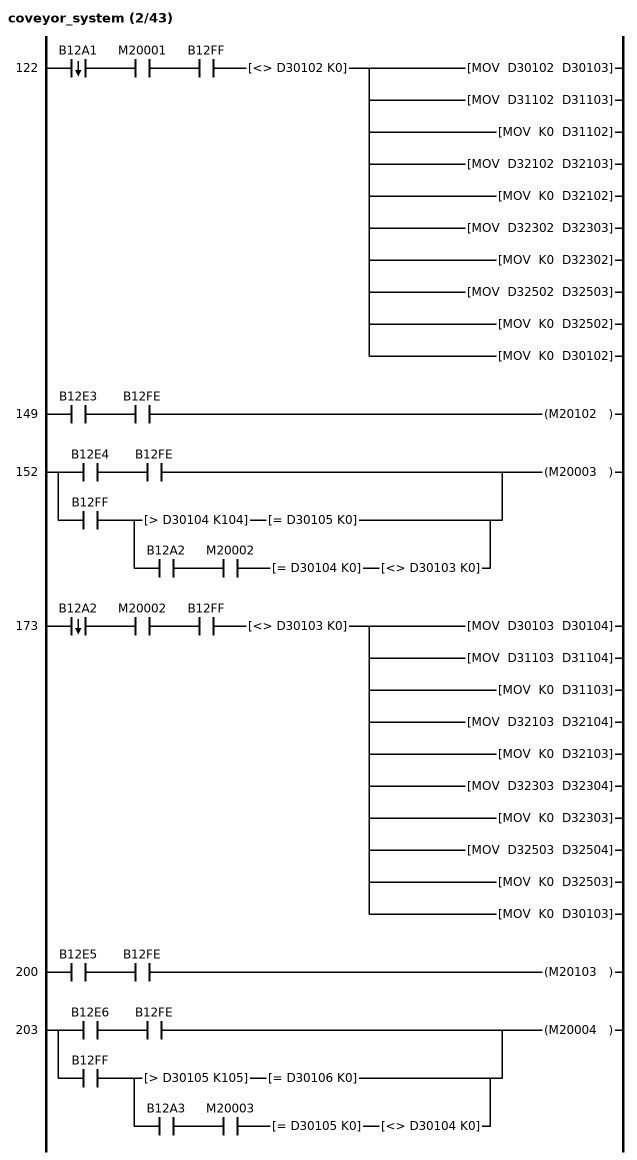
[picture p168: ladder of coveyor_system, rungs at steps 122 to 203]
122   LDF     B12A1
      AND     M20001
      AND     B12FF
      AND<>   D30102 K0
      MOV     D30102 D30103
      MOV     D31102 D31103
      MOV     K0 D31102
      MOV     D32102 D32103
      MOV     K0 D32102
      MOV     D32302 D32303
      MOV     K0 D32302
      MOV     D32502 D32503
      MOV     K0 D32502
      MOV     K0 D30102
149   LD      B12E3
      AND     B12FE
      OUT     M20102
152   LD      B12E4
      AND     B12FE
      LD      B12FF
      LD>     D30104 K104
      AND=    D30105 K0
      LD      B12A2
      AND     M20002
      AND=    D30104 K0
      AND<>   D30103 K0
      ORB
      ANB
      ORB
      OUT     M20003
173   LDF     B12A2
      AND     M20002
      AND     B12FF
      AND<>   D30103 K0
      MOV     D30103 D30104
      MOV     D31103 D31104
      MOV     K0 D31103
      MOV     D32103 D32104
      MOV     K0 D32103
      MOV     D32303 D32304
      MOV     K0 D32303
      MOV     D32503 D32504
      MOV     K0 D32503
      MOV     K0 D30103
200   LD      B12E5
      AND     B12FE
      OUT     M20103
203   LD      B12E6
      AND     B12FE
      LD      B12FF
      LD>     D30105 K105
      AND=    D30106 K0
      LD      B12A3
      AND     M20003
      AND=    D30105 K0
      AND<>   D30104 K0
      ORB
      ANB
      ORB
      OUT     M20004
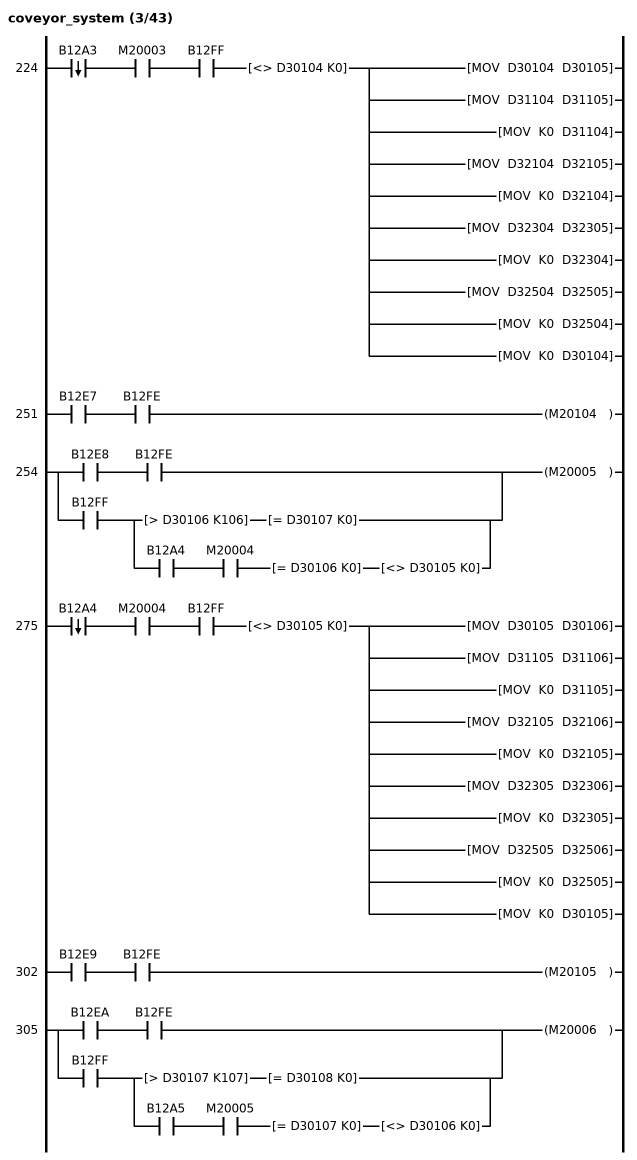
224   LDF     B12A3
      AND     M20003
      AND     B12FF
      AND<>   D30104 K0
      MOV     D30104 D30105
      MOV     D31104 D31105
      MOV     K0 D31104
      MOV     D32104 D32105
      MOV     K0 D32104
      MOV     D32304 D32305
      MOV     K0 D32304
      MOV     D32504 D32505
      MOV     K0 D32504
      MOV     K0 D30104
251   LD      B12E7
      AND     B12FE
      OUT     M20104
254   LD      B12E8
      AND     B12FE
      LD      B12FF
      LD>     D30106 K106
      AND=    D30107 K0
      LD      B12A4
      AND     M20004
      AND=    D30106 K0
      AND<>   D30105 K0
      ORB
      ANB
      ORB
      OUT     M20005
275   LDF     B12A4
      AND     M20004
      AND     B12FF
      AND<>   D30105 K0
      MOV     D30105 D30106
      MOV     D31105 D31106
      MOV     K0 D31105
      MOV     D32105 D32106
      MOV     K0 D32105
      MOV     D32305 D32306
      MOV     K0 D32305
      MOV     D32505 D32506
      MOV     K0 D32505
      MOV     K0 D30105
302   LD      B12E9
      AND     B12FE
      OUT     M20105
305   LD      B12EA
      AND     B12FE
      LD      B12FF
      LD>     D30107 K107
      AND=    D30108 K0
      LD      B12A5
      AND     M20005
      AND=    D30107 K0
      AND<>   D30106 K0
      ORB
      ANB
      ORB
      OUT     M20006
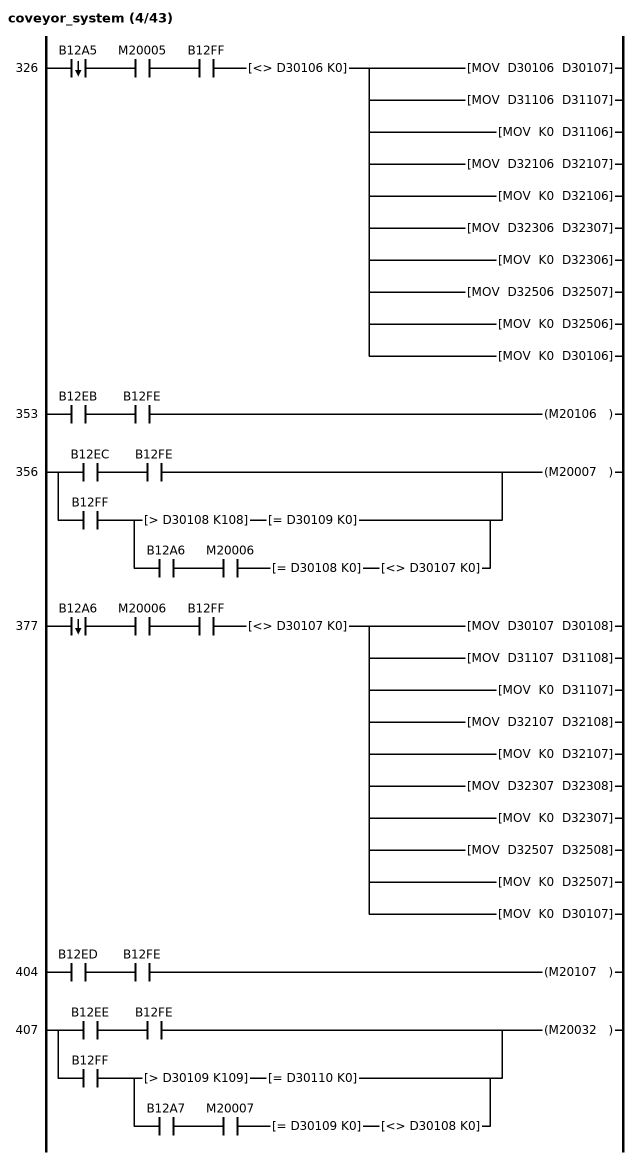
326   LDF     B12A5
      AND     M20005
      AND     B12FF
      AND<>   D30106 K0
      MOV     D30106 D30107
      MOV     D31106 D31107
      MOV     K0 D31106
      MOV     D32106 D32107
      MOV     K0 D32106
      MOV     D32306 D32307
      MOV     K0 D32306
      MOV     D32506 D32507
      MOV     K0 D32506
      MOV     K0 D30106
353   LD      B12EB
      AND     B12FE
      OUT     M20106
356   LD      B12EC
      AND     B12FE
      LD      B12FF
      LD>     D30108 K108
      AND=    D30109 K0
      LD      B12A6
      AND     M20006
      AND=    D30108 K0
      AND<>   D30107 K0
      ORB
      ANB
      ORB
      OUT     M20007
377   LDF     B12A6
      AND     M20006
      AND     B12FF
      AND<>   D30107 K0
      MOV     D30107 D30108
      MOV     D31107 D31108
      MOV     K0 D31107
      MOV     D32107 D32108
      MOV     K0 D32107
      MOV     D32307 D32308
      MOV     K0 D32307
      MOV     D32507 D32508
      MOV     K0 D32507
      MOV     K0 D30107
404   LD      B12ED
      AND     B12FE
      OUT     M20107
407   LD      B12EE
      AND     B12FE
      LD      B12FF
      LD>     D30109 K109
      AND=    D30110 K0
      LD      B12A7
      AND     M20007
      AND=    D30109 K0
      AND<>   D30108 K0
      ORB
      ANB
      ORB
      OUT     M20032
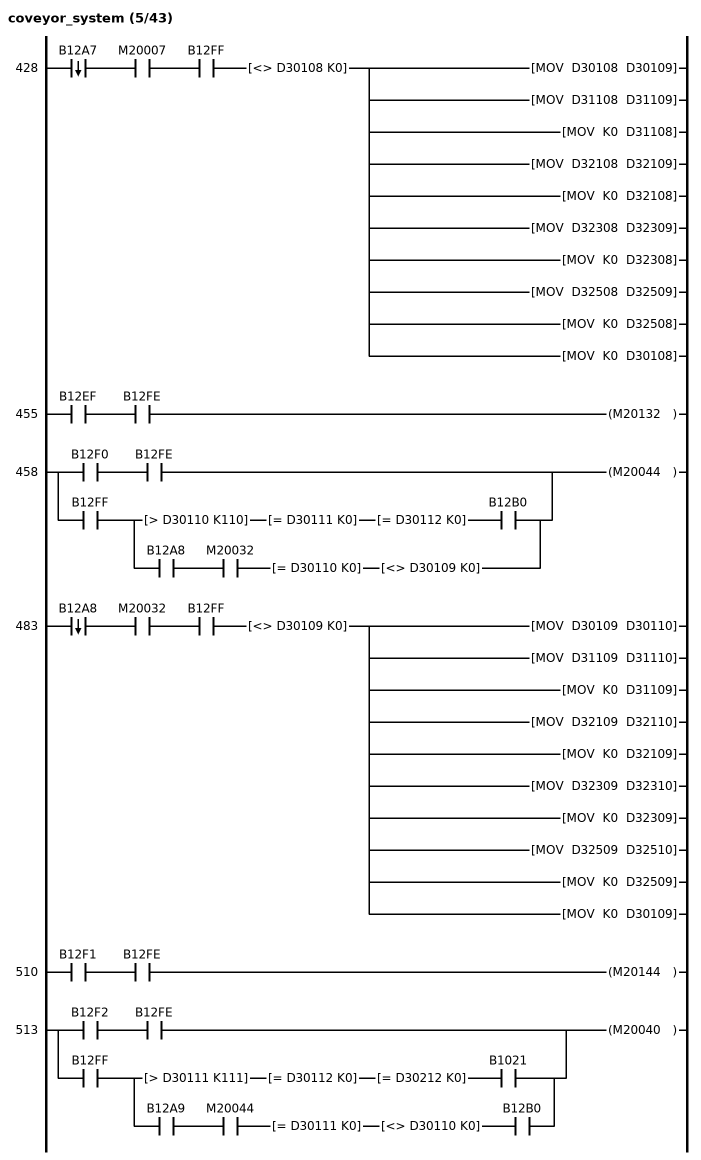
428   LDF     B12A7
      AND     M20007
      AND     B12FF
      AND<>   D30108 K0
      MOV     D30108 D30109
      MOV     D31108 D31109
      MOV     K0 D31108
      MOV     D32108 D32109
      MOV     K0 D32108
      MOV     D32308 D32309
      MOV     K0 D32308
      MOV     D32508 D32509
      MOV     K0 D32508
      MOV     K0 D30108
455   LD      B12EF
      AND     B12FE
      OUT     M20132
458   LD      B12F0
      AND     B12FE
      LD      B12FF
      LD>     D30110 K110
      AND=    D30111 K0
      AND=    D30112 K0
      AND     B12B0
      LD      B12A8
      AND     M20032
      AND=    D30110 K0
      AND<>   D30109 K0
      ORB
      ANB
      ORB
      OUT     M20044
483   LDF     B12A8
      AND     M20032
      AND     B12FF
      AND<>   D30109 K0
      MOV     D30109 D30110
      MOV     D31109 D31110
      MOV     K0 D31109
      MOV     D32109 D32110
      MOV     K0 D32109
      MOV     D32309 D32310
      MOV     K0 D32309
      MOV     D32509 D32510
      MOV     K0 D32509
      MOV     K0 D30109
510   LD      B12F1
      AND     B12FE
      OUT     M20144
513   LD      B12F2
      AND     B12FE
      LD      B12FF
      LD>     D30111 K111
      AND=    D30112 K0
      AND=    D30212 K0
      AND     B1021
      LD      B12A9
      AND     M20044
      AND=    D30111 K0
      AND<>   D30110 K0
      AND     B12B0
      ORB
      ANB
      ORB
      OUT     M20040
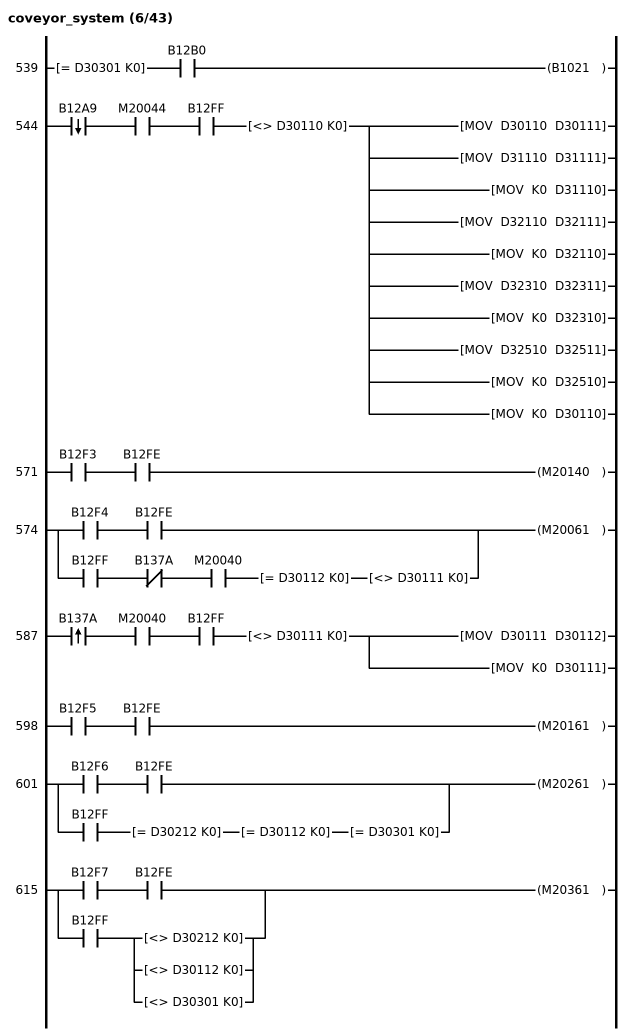
539   LD=     D30301 K0
      AND     B12B0
      OUT     B1021
544   LDF     B12A9
      AND     M20044
      AND     B12FF
      AND<>   D30110 K0
      MOV     D30110 D30111
      MOV     D31110 D31111
      MOV     K0 D31110
      MOV     D32110 D32111
      MOV     K0 D32110
      MOV     D32310 D32311
      MOV     K0 D32310
      MOV     D32510 D32511
      MOV     K0 D32510
      MOV     K0 D30110
571   LD      B12F3
      AND     B12FE
      OUT     M20140
574   LD      B12F4
      AND     B12FE
      LD      B12FF
      ANI     B137A
      AND     M20040
      AND=    D30112 K0
      AND<>   D30111 K0
      ORB
      OUT     M20061
587   LDP     B137A
      AND     M20040
      AND     B12FF
      AND<>   D30111 K0
      MOV     D30111 D30112
      MOV     K0 D30111
598   LD      B12F5
      AND     B12FE
      OUT     M20161
601   LD      B12F6
      AND     B12FE
      LD      B12FF
      AND=    D30212 K0
      AND=    D30112 K0
      AND=    D30301 K0
      ORB
      OUT     M20261
615   LD      B12F7
      AND     B12FE
      LD      B12FF
      LD<>    D30212 K0
      OR<>    D30112 K0
      OR<>    D30301 K0
      ANB
      ORB
      OUT     M20361
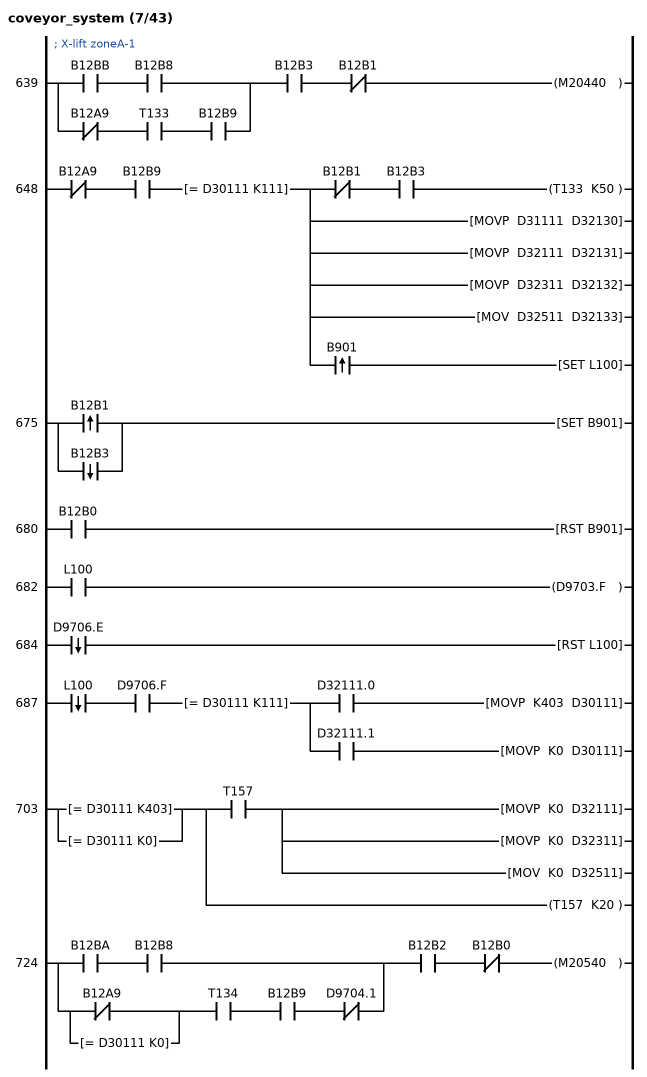
; X-lift zoneA-1
639   LD      B12BB
      AND     B12B8
      LDI     B12A9
      AND     T133
      AND     B12B9
      ORB
      AND     B12B3
      ANI     B12B1
      OUT     M20440
648   LDI     B12A9
      AND     B12B9
      AND=    D30111 K111
      MPS
      ANI     B12B1
      AND     B12B3
      OUT     T133 K50
      MPP
      MOVP    D31111 D32130
      MOVP    D32111 D32131
      MOVP    D32311 D32132
      MOV     D32511 D32133
      ANDP    B901
      SET     L100
675   LDP     B12B1
      ORF     B12B3
      SET     B901
680   LD      B12B0
      RST     B901
682   LD      L100
      OUT     D9703.F
684   LDF     D9706.E
      RST     L100
687   LDF     L100
      AND     D9706.F
      AND=    D30111 K111
      MPS
      AND     D32111.0
      MOVP    K403 D30111
      MPP
      AND     D32111.1
      MOVP    K0 D30111
703   LD=     D30111 K403
      OR=     D30111 K0
      MPS
      AND     T157
      MOVP    K0 D32111
      MOVP    K0 D32311
      MOV     K0 D32511
      MPP
      OUT     T157 K20
724   LD      B12BA
      AND     B12B8
      LDI     B12A9
      OR=     D30111 K0
      AND     T134
      AND     B12B9
      ANI     D9704.1
      ORB
      AND     B12B2
      ANI     B12B0
      OUT     M20540
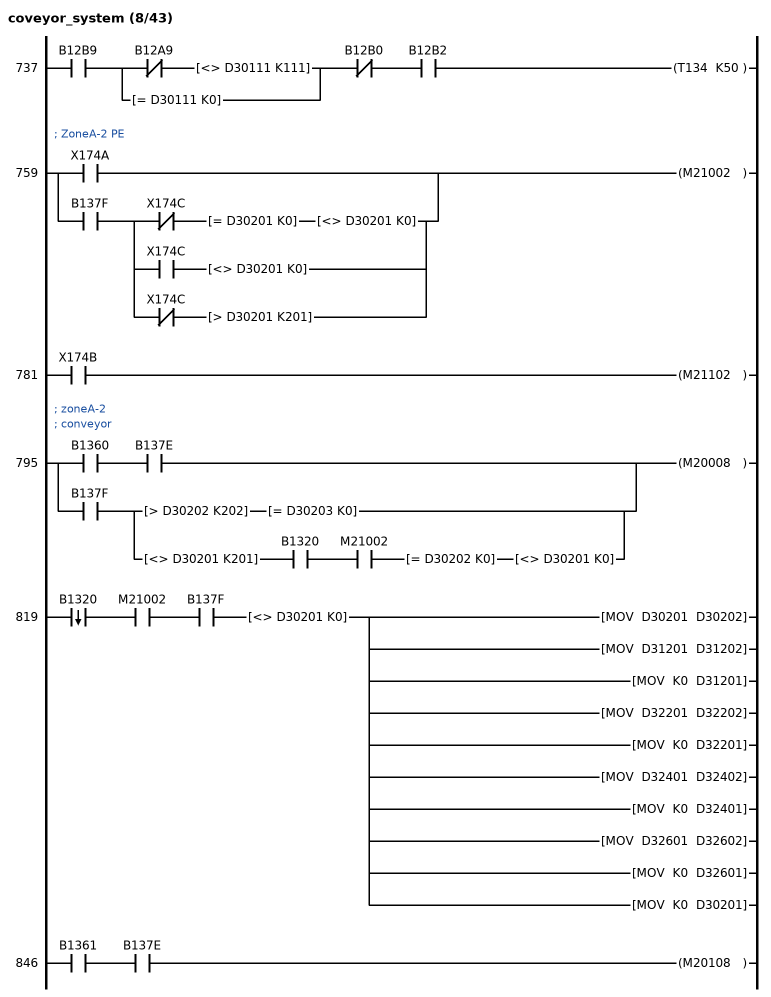
737   LD      B12B9
      LDI     B12A9
      AND<>   D30111 K111
      OR=     D30111 K0
      ANB
      ANI     B12B0
      AND     B12B2
      OUT     T134 K50
; ZoneA-2 PE
759   LD      X174A
      LD      B137F
      LDI     X174C
      AND=    D30201 K0
      AND<>   D30201 K0
      LD      X174C
      AND<>   D30201 K0
      ORB
      LDI     X174C
      AND>    D30201 K201
      ORB
      ANB
      ORB
      OUT     M21002
781   LD      X174B
      OUT     M21102
; zoneA-2
; conveyor
795   LD      B1360
      AND     B137E
      LD      B137F
      LD>     D30202 K202
      AND=    D30203 K0
      LD<>    D30201 K201
      AND     B1320
      AND     M21002
      AND=    D30202 K0
      AND<>   D30201 K0
      ORB
      ANB
      ORB
      OUT     M20008
819   LDF     B1320
      AND     M21002
      AND     B137F
      AND<>   D30201 K0
      MOV     D30201 D30202
      MOV     D31201 D31202
      MOV     K0 D31201
      MOV     D32201 D32202
      MOV     K0 D32201
      MOV     D32401 D32402
      MOV     K0 D32401
      MOV     D32601 D32602
      MOV     K0 D32601
      MOV     K0 D30201
846   LD      B1361
      AND     B137E
      OUT     M20108
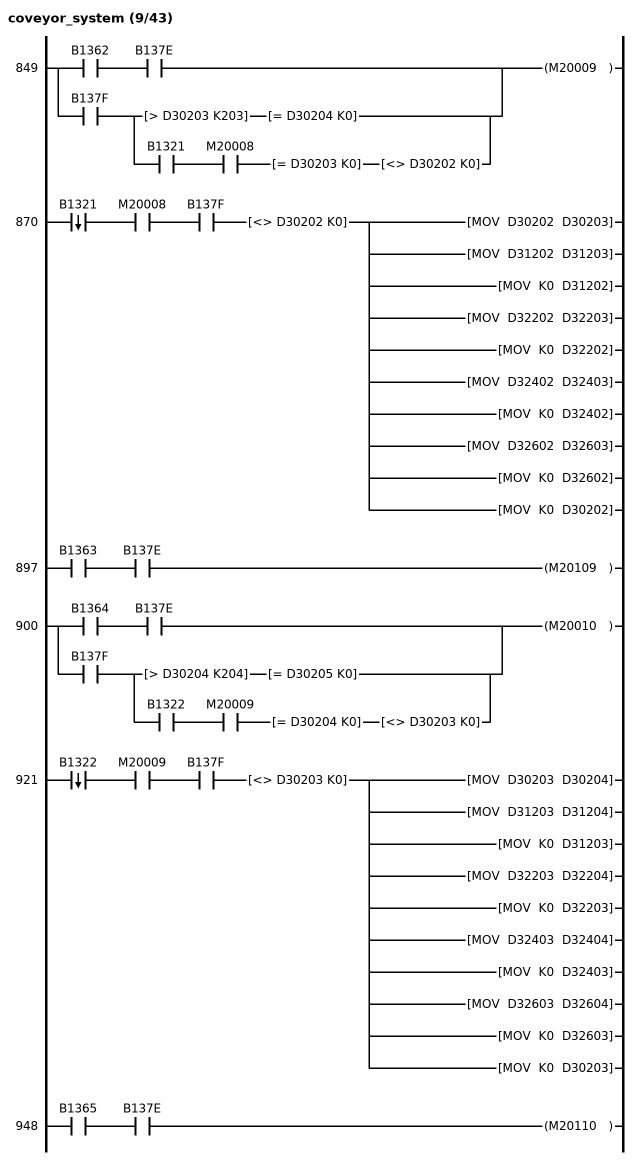
849   LD      B1362
      AND     B137E
      LD      B137F
      LD>     D30203 K203
      AND=    D30204 K0
      LD      B1321
      AND     M20008
      AND=    D30203 K0
      AND<>   D30202 K0
      ORB
      ANB
      ORB
      OUT     M20009
870   LDF     B1321
      AND     M20008
      AND     B137F
      AND<>   D30202 K0
      MOV     D30202 D30203
      MOV     D31202 D31203
      MOV     K0 D31202
      MOV     D32202 D32203
      MOV     K0 D32202
      MOV     D32402 D32403
      MOV     K0 D32402
      MOV     D32602 D32603
      MOV     K0 D32602
      MOV     K0 D30202
897   LD      B1363
      AND     B137E
      OUT     M20109
900   LD      B1364
      AND     B137E
      LD      B137F
      LD>     D30204 K204
      AND=    D30205 K0
      LD      B1322
      AND     M20009
      AND=    D30204 K0
      AND<>   D30203 K0
      ORB
      ANB
      ORB
      OUT     M20010
921   LDF     B1322
      AND     M20009
      AND     B137F
      AND<>   D30203 K0
      MOV     D30203 D30204
      MOV     D31203 D31204
      MOV     K0 D31203
      MOV     D32203 D32204
      MOV     K0 D32203
      MOV     D32403 D32404
      MOV     K0 D32403
      MOV     D32603 D32604
      MOV     K0 D32603
      MOV     K0 D30203
948   LD      B1365
      AND     B137E
      OUT     M20110
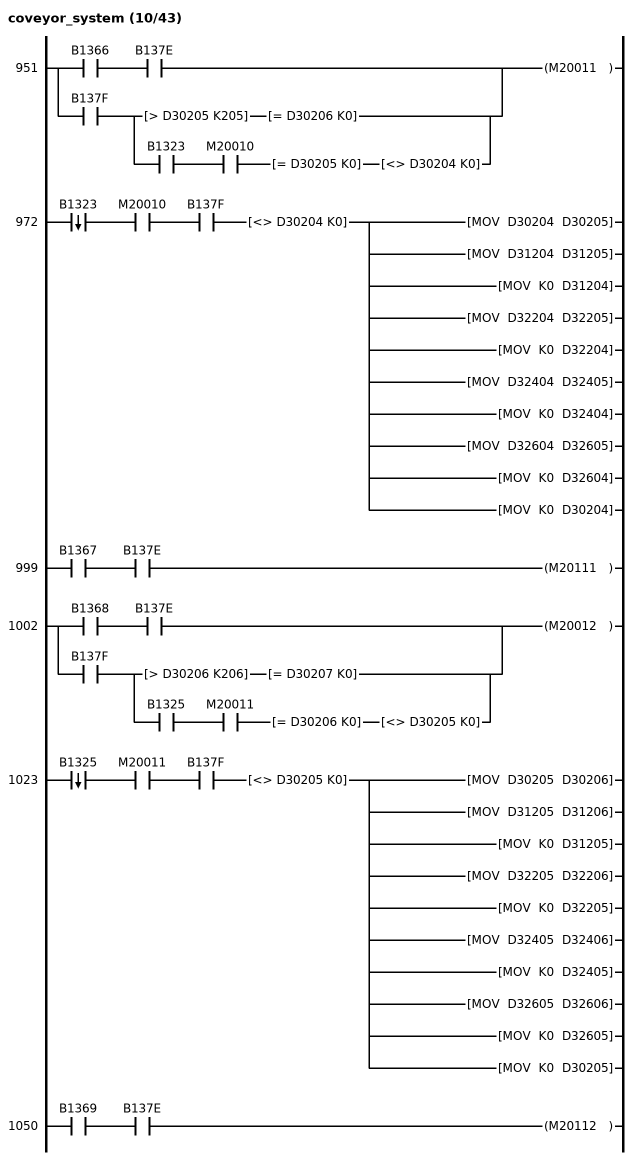
951   LD      B1366
      AND     B137E
      LD      B137F
      LD>     D30205 K205
      AND=    D30206 K0
      LD      B1323
      AND     M20010
      AND=    D30205 K0
      AND<>   D30204 K0
      ORB
      ANB
      ORB
      OUT     M20011
972   LDF     B1323
      AND     M20010
      AND     B137F
      AND<>   D30204 K0
      MOV     D30204 D30205
      MOV     D31204 D31205
      MOV     K0 D31204
      MOV     D32204 D32205
      MOV     K0 D32204
      MOV     D32404 D32405
      MOV     K0 D32404
      MOV     D32604 D32605
      MOV     K0 D32604
      MOV     K0 D30204
999   LD      B1367
      AND     B137E
      OUT     M20111
1002  LD      B1368
      AND     B137E
      LD      B137F
      LD>     D30206 K206
      AND=    D30207 K0
      LD      B1325
      AND     M20011
      AND=    D30206 K0
      AND<>   D30205 K0
      ORB
      ANB
      ORB
      OUT     M20012
1023  LDF     B1325
      AND     M20011
      AND     B137F
      AND<>   D30205 K0
      MOV     D30205 D30206
      MOV     D31205 D31206
      MOV     K0 D31205
      MOV     D32205 D32206
      MOV     K0 D32205
      MOV     D32405 D32406
      MOV     K0 D32405
      MOV     D32605 D32606
      MOV     K0 D32605
      MOV     K0 D30205
1050  LD      B1369
      AND     B137E
      OUT     M20112
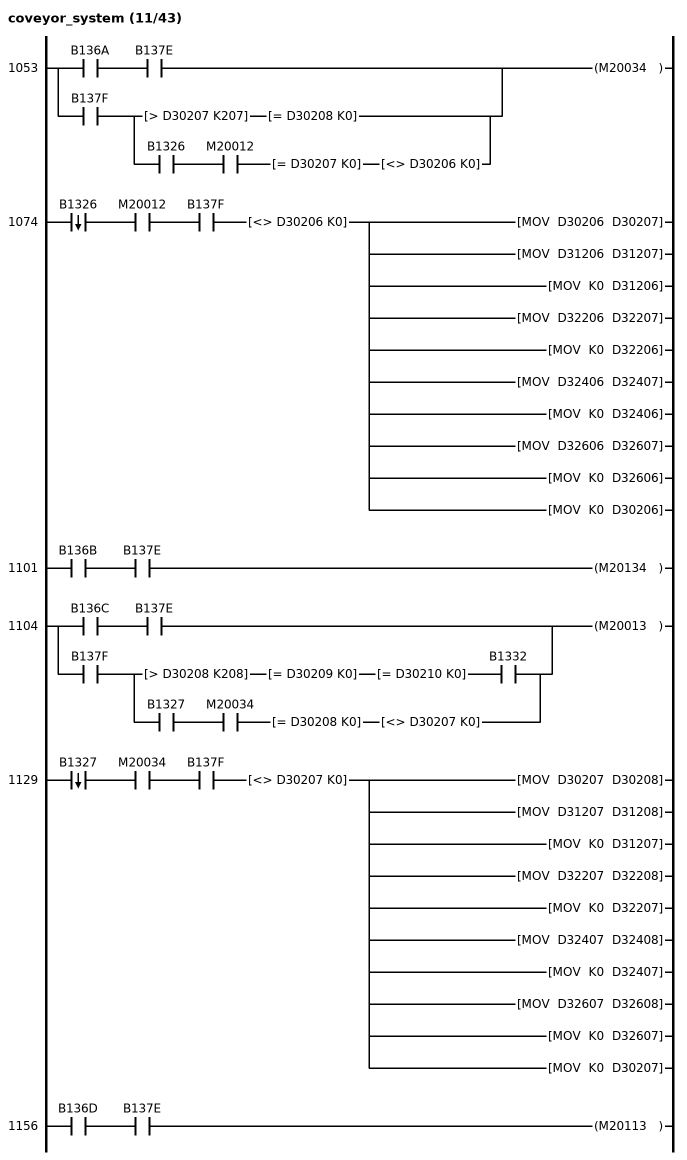
1053  LD      B136A
      AND     B137E
      LD      B137F
      LD>     D30207 K207
      AND=    D30208 K0
      LD      B1326
      AND     M20012
      AND=    D30207 K0
      AND<>   D30206 K0
      ORB
      ANB
      ORB
      OUT     M20034
1074  LDF     B1326
      AND     M20012
      AND     B137F
      AND<>   D30206 K0
      MOV     D30206 D30207
      MOV     D31206 D31207
      MOV     K0 D31206
      MOV     D32206 D32207
      MOV     K0 D32206
      MOV     D32406 D32407
      MOV     K0 D32406
      MOV     D32606 D32607
      MOV     K0 D32606
      MOV     K0 D30206
1101  LD      B136B
      AND     B137E
      OUT     M20134
1104  LD      B136C
      AND     B137E
      LD      B137F
      LD>     D30208 K208
      AND=    D30209 K0
      AND=    D30210 K0
      AND     B1332
      LD      B1327
      AND     M20034
      AND=    D30208 K0
      AND<>   D30207 K0
      ORB
      ANB
      ORB
      OUT     M20013
1129  LDF     B1327
      AND     M20034
      AND     B137F
      AND<>   D30207 K0
      MOV     D30207 D30208
      MOV     D31207 D31208
      MOV     K0 D31207
      MOV     D32207 D32208
      MOV     K0 D32207
      MOV     D32407 D32408
      MOV     K0 D32407
      MOV     D32607 D32608
      MOV     K0 D32607
      MOV     K0 D30207
1156  LD      B136D
      AND     B137E
      OUT     M20113
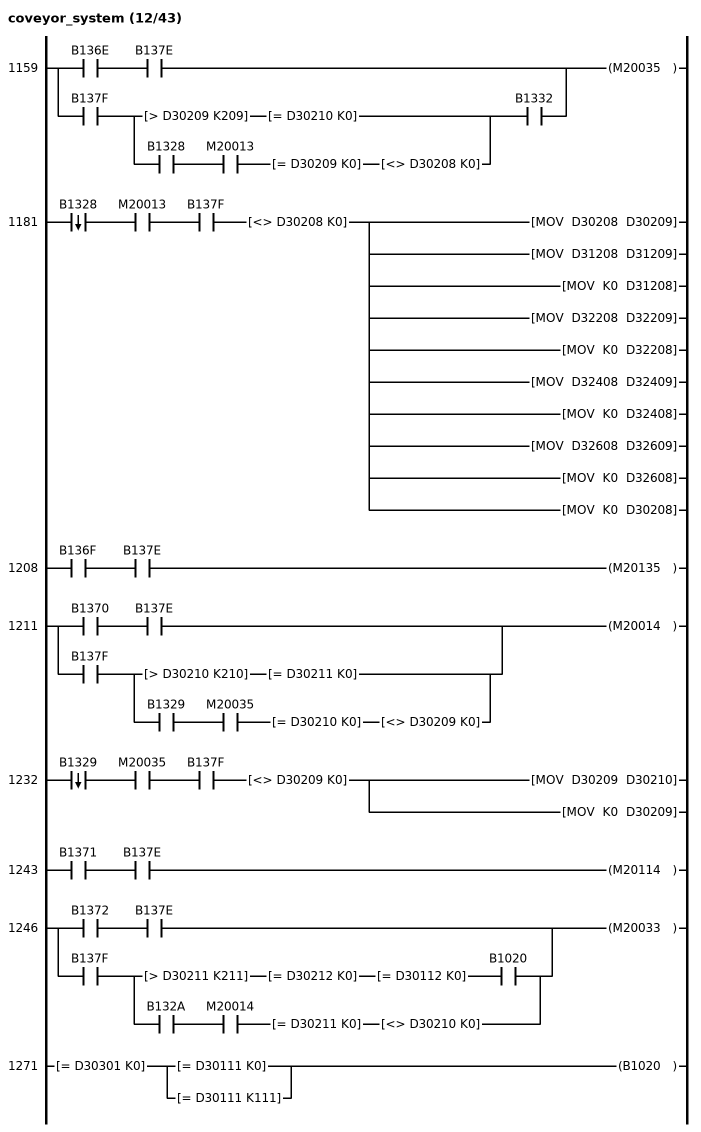
1159  LD      B136E
      AND     B137E
      LD      B137F
      LD>     D30209 K209
      AND=    D30210 K0
      LD      B1328
      AND     M20013
      AND=    D30209 K0
      AND<>   D30208 K0
      ORB
      ANB
      AND     B1332
      ORB
      OUT     M20035
1181  LDF     B1328
      AND     M20013
      AND     B137F
      AND<>   D30208 K0
      MOV     D30208 D30209
      MOV     D31208 D31209
      MOV     K0 D31208
      MOV     D32208 D32209
      MOV     K0 D32208
      MOV     D32408 D32409
      MOV     K0 D32408
      MOV     D32608 D32609
      MOV     K0 D32608
      MOV     K0 D30208
1208  LD      B136F
      AND     B137E
      OUT     M20135
1211  LD      B1370
      AND     B137E
      LD      B137F
      LD>     D30210 K210
      AND=    D30211 K0
      LD      B1329
      AND     M20035
      AND=    D30210 K0
      AND<>   D30209 K0
      ORB
      ANB
      ORB
      OUT     M20014
1232  LDF     B1329
      AND     M20035
      AND     B137F
      AND<>   D30209 K0
      MOV     D30209 D30210
      MOV     K0 D30209
1243  LD      B1371
      AND     B137E
      OUT     M20114
1246  LD      B1372
      AND     B137E
      LD      B137F
      LD>     D30211 K211
      AND=    D30212 K0
      AND=    D30112 K0
      AND     B1020
      LD      B132A
      AND     M20014
      AND=    D30211 K0
      AND<>   D30210 K0
      ORB
      ANB
      ORB
      OUT     M20033
1271  LD=     D30301 K0
      LD=     D30111 K0
      OR=     D30111 K111
      ANB
      OUT     B1020
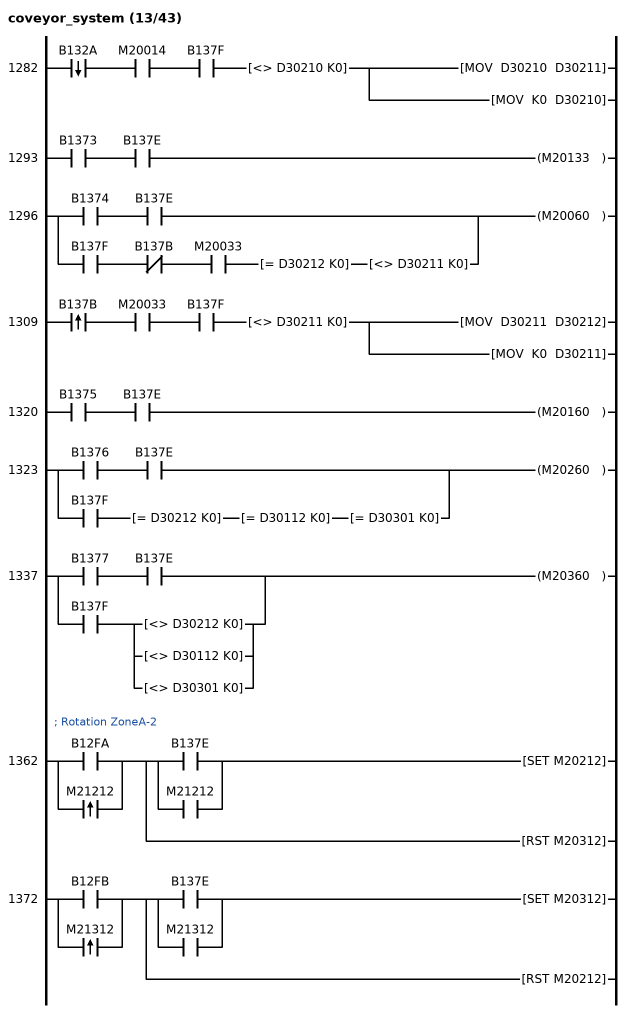
1282  LDF     B132A
      AND     M20014
      AND     B137F
      AND<>   D30210 K0
      MOV     D30210 D30211
      MOV     K0 D30210
1293  LD      B1373
      AND     B137E
      OUT     M20133
1296  LD      B1374
      AND     B137E
      LD      B137F
      ANI     B137B
      AND     M20033
      AND=    D30212 K0
      AND<>   D30211 K0
      ORB
      OUT     M20060
1309  LDP     B137B
      AND     M20033
      AND     B137F
      AND<>   D30211 K0
      MOV     D30211 D30212
      MOV     K0 D30211
1320  LD      B1375
      AND     B137E
      OUT     M20160
1323  LD      B1376
      AND     B137E
      LD      B137F
      AND=    D30212 K0
      AND=    D30112 K0
      AND=    D30301 K0
      ORB
      OUT     M20260
1337  LD      B1377
      AND     B137E
      LD      B137F
      LD<>    D30212 K0
      OR<>    D30112 K0
      OR<>    D30301 K0
      ANB
      ORB
      OUT     M20360
; Rotation ZoneA-2
1362  LD      B12FA
      ORP     M21212
      MPS
      LD      B137E
      OR      M21212
      ANB
      SET     M20212
      MPP
      RST     M20312
1372  LD      B12FB
      ORP     M21312
      MPS
      LD      B137E
      OR      M21312
      ANB
      SET     M20312
      MPP
      RST     M20212
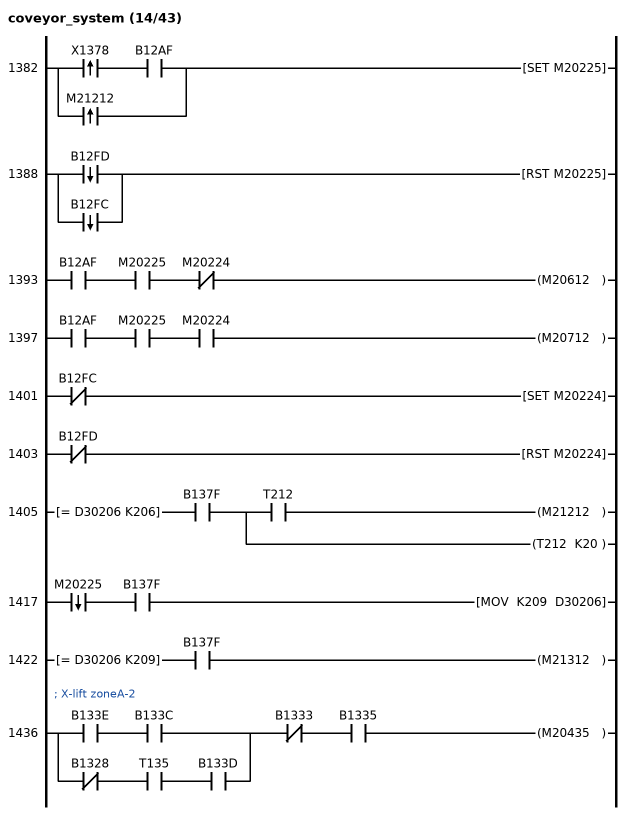
1382  LDP     X1378
      AND     B12AF
      ORP     M21212
      SET     M20225
1388  LDF     B12FD
      ORF     B12FC
      RST     M20225
1393  LD      B12AF
      AND     M20225
      ANI     M20224
      OUT     M20612
1397  LD      B12AF
      AND     M20225
      AND     M20224
      OUT     M20712
1401  LDI     B12FC
      SET     M20224
1403  LDI     B12FD
      RST     M20224
1405  LD=     D30206 K206
      AND     B137F
      MPS
      AND     T212
      OUT     M21212
      MPP
      OUT     T212 K20
1417  LDF     M20225
      AND     B137F
      MOV     K209 D30206
1422  LD=     D30206 K209
      AND     B137F
      OUT     M21312
; X-lift zoneA-2
1436  LD      B133E
      AND     B133C
      LDI     B1328
      AND     T135
      AND     B133D
      ORB
      ANI     B1333
      AND     B1335
      OUT     M20435
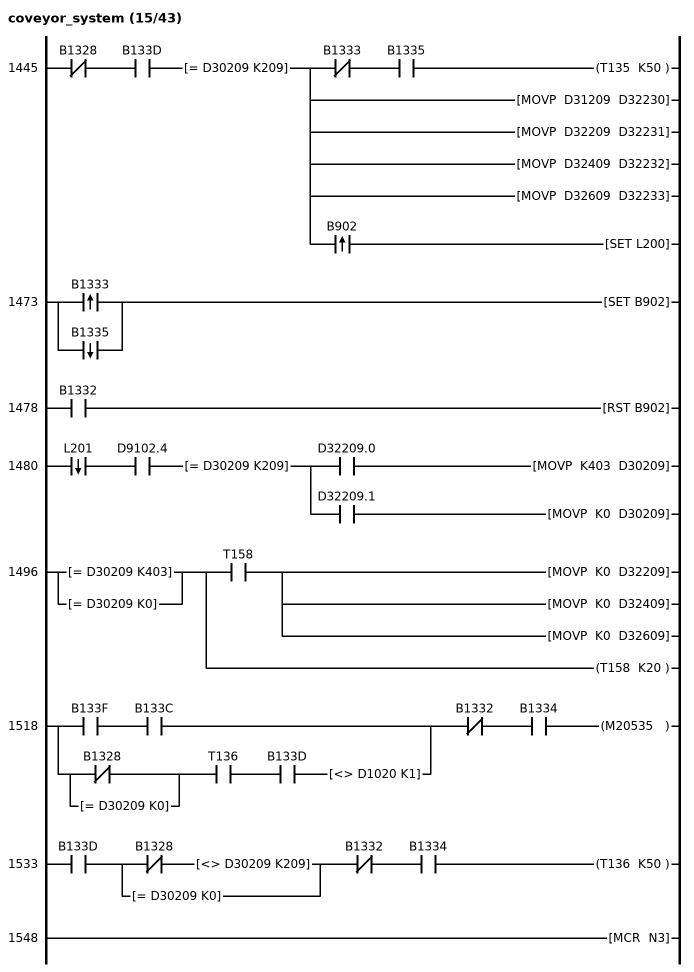
1445  LDI     B1328
      AND     B133D
      AND=    D30209 K209
      MPS
      ANI     B1333
      AND     B1335
      OUT     T135 K50
      MPP
      MOVP    D31209 D32230
      MOVP    D32209 D32231
      MOVP    D32409 D32232
      MOVP    D32609 D32233
      ANDP    B902
      SET     L200
1473  LDP     B1333
      ORF     B1335
      SET     B902
1478  LD      B1332
      RST     B902
1480  LDF     L201
      AND     D9102.4
      AND=    D30209 K209
      MPS
      AND     D32209.0
      MOVP    K403 D30209
      MPP
      AND     D32209.1
      MOVP    K0 D30209
1496  LD=     D30209 K403
      OR=     D30209 K0
      MPS
      AND     T158
      MOVP    K0 D32209
      MOVP    K0 D32409
      MOVP    K0 D32609
      MPP
      OUT     T158 K20
1518  LD      B133F
      AND     B133C
      LDI     B1328
      OR=     D30209 K0
      AND     T136
      AND     B133D
      AND<>   D1020 K1
      ORB
      ANI     B1332
      AND     B1334
      OUT     M20535
1533  LD      B133D
      LDI     B1328
      AND<>   D30209 K209
      OR=     D30209 K0
      ANB
      ANI     B1332
      AND     B1334
      OUT     T136 K50
1548  MCR     N3
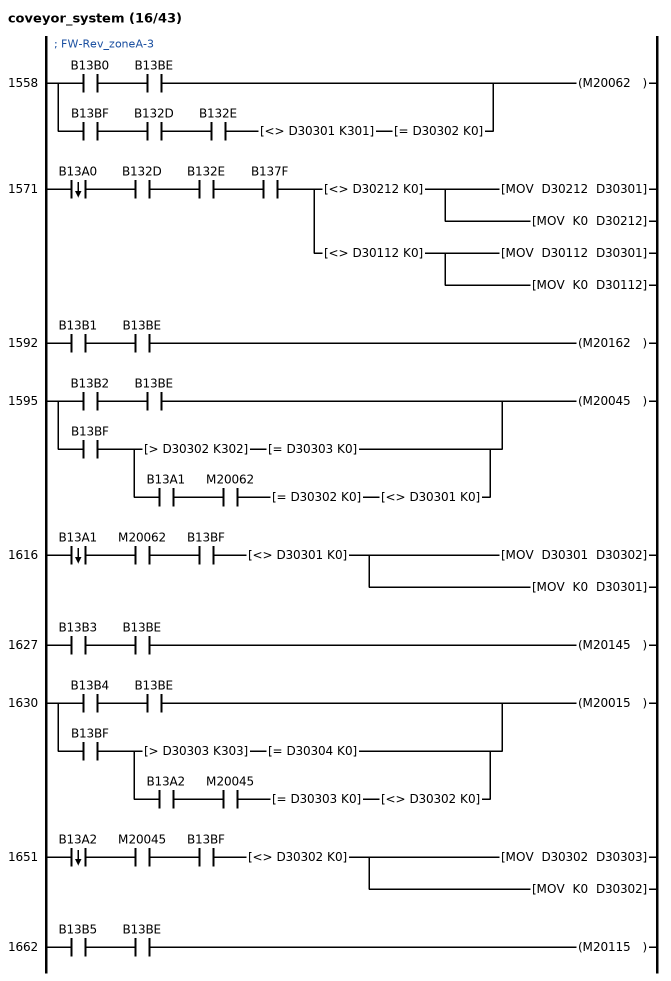
; FW-Rev_zoneA-3
1558  LD      B13B0
      AND     B13BE
      LD      B13BF
      AND     B132D
      AND     B132E
      AND<>   D30301 K301
      AND=    D30302 K0
      ORB
      OUT     M20062
1571  LDF     B13A0
      AND     B132D
      AND     B132E
      AND     B137F
      MPS
      AND<>   D30212 K0
      MOV     D30212 D30301
      MOV     K0 D30212
      MPP
      AND<>   D30112 K0
      MOV     D30112 D30301
      MOV     K0 D30112
1592  LD      B13B1
      AND     B13BE
      OUT     M20162
1595  LD      B13B2
      AND     B13BE
      LD      B13BF
      LD>     D30302 K302
      AND=    D30303 K0
      LD      B13A1
      AND     M20062
      AND=    D30302 K0
      AND<>   D30301 K0
      ORB
      ANB
      ORB
      OUT     M20045
1616  LDF     B13A1
      AND     M20062
      AND     B13BF
      AND<>   D30301 K0
      MOV     D30301 D30302
      MOV     K0 D30301
1627  LD      B13B3
      AND     B13BE
      OUT     M20145
1630  LD      B13B4
      AND     B13BE
      LD      B13BF
      LD>     D30303 K303
      AND=    D30304 K0
      LD      B13A2
      AND     M20045
      AND=    D30303 K0
      AND<>   D30302 K0
      ORB
      ANB
      ORB
      OUT     M20015
1651  LDF     B13A2
      AND     M20045
      AND     B13BF
      AND<>   D30302 K0
      MOV     D30302 D30303
      MOV     K0 D30302
1662  LD      B13B5
      AND     B13BE
      OUT     M20115
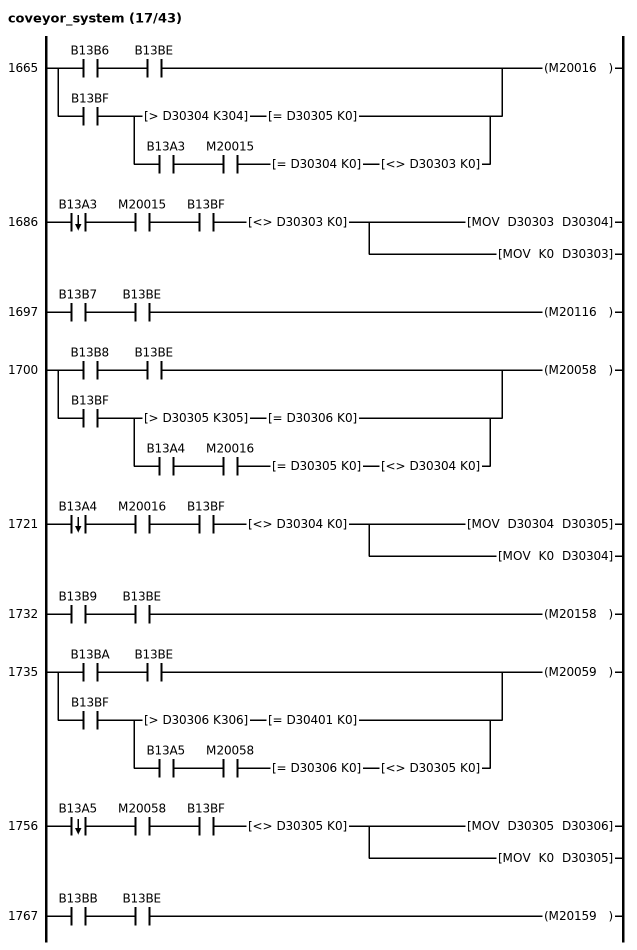
1665  LD      B13B6
      AND     B13BE
      LD      B13BF
      LD>     D30304 K304
      AND=    D30305 K0
      LD      B13A3
      AND     M20015
      AND=    D30304 K0
      AND<>   D30303 K0
      ORB
      ANB
      ORB
      OUT     M20016
1686  LDF     B13A3
      AND     M20015
      AND     B13BF
      AND<>   D30303 K0
      MOV     D30303 D30304
      MOV     K0 D30303
1697  LD      B13B7
      AND     B13BE
      OUT     M20116
1700  LD      B13B8
      AND     B13BE
      LD      B13BF
      LD>     D30305 K305
      AND=    D30306 K0
      LD      B13A4
      AND     M20016
      AND=    D30305 K0
      AND<>   D30304 K0
      ORB
      ANB
      ORB
      OUT     M20058
1721  LDF     B13A4
      AND     M20016
      AND     B13BF
      AND<>   D30304 K0
      MOV     D30304 D30305
      MOV     K0 D30304
1732  LD      B13B9
      AND     B13BE
      OUT     M20158
1735  LD      B13BA
      AND     B13BE
      LD      B13BF
      LD>     D30306 K306
      AND=    D30401 K0
      LD      B13A5
      AND     M20058
      AND=    D30306 K0
      AND<>   D30305 K0
      ORB
      ANB
      ORB
      OUT     M20059
1756  LDF     B13A5
      AND     M20058
      AND     B13BF
      AND<>   D30305 K0
      MOV     D30305 D30306
      MOV     K0 D30305
1767  LD      B13BB
      AND     B13BE
      OUT     M20159
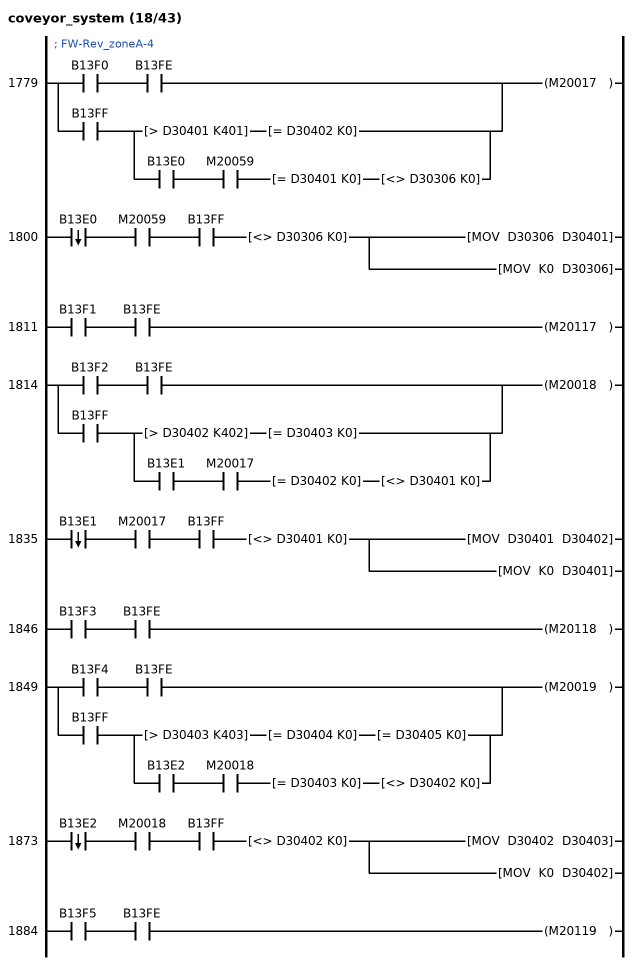
; FW-Rev_zoneA-4
1779  LD      B13F0
      AND     B13FE
      LD      B13FF
      LD>     D30401 K401
      AND=    D30402 K0
      LD      B13E0
      AND     M20059
      AND=    D30401 K0
      AND<>   D30306 K0
      ORB
      ANB
      ORB
      OUT     M20017
1800  LDF     B13E0
      AND     M20059
      AND     B13FF
      AND<>   D30306 K0
      MOV     D30306 D30401
      MOV     K0 D30306
1811  LD      B13F1
      AND     B13FE
      OUT     M20117
1814  LD      B13F2
      AND     B13FE
      LD      B13FF
      LD>     D30402 K402
      AND=    D30403 K0
      LD      B13E1
      AND     M20017
      AND=    D30402 K0
      AND<>   D30401 K0
      ORB
      ANB
      ORB
      OUT     M20018
1835  LDF     B13E1
      AND     M20017
      AND     B13FF
      AND<>   D30401 K0
      MOV     D30401 D30402
      MOV     K0 D30401
1846  LD      B13F3
      AND     B13FE
      OUT     M20118
1849  LD      B13F4
      AND     B13FE
      LD      B13FF
      LD>     D30403 K403
      AND=    D30404 K0
      AND=    D30405 K0
      LD      B13E2
      AND     M20018
      AND=    D30403 K0
      AND<>   D30402 K0
      ORB
      ANB
      ORB
      OUT     M20019
1873  LDF     B13E2
      AND     M20018
      AND     B13FF
      AND<>   D30402 K0
      MOV     D30402 D30403
      MOV     K0 D30402
1884  LD      B13F5
      AND     B13FE
      OUT     M20119
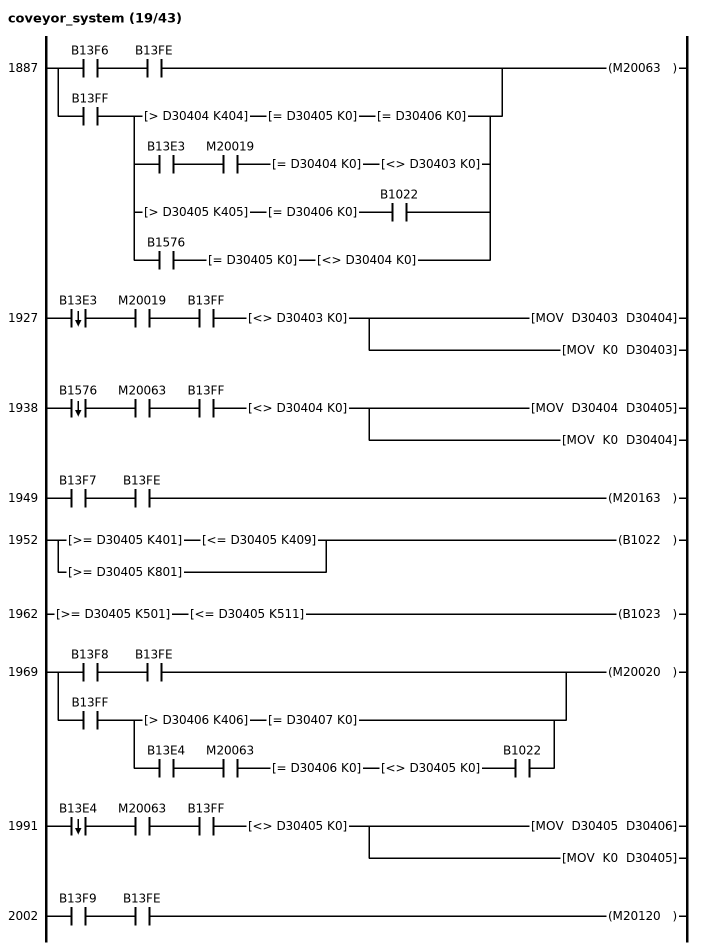
1887  LD      B13F6
      AND     B13FE
      LD      B13FF
      LD>     D30404 K404
      AND=    D30405 K0
      AND=    D30406 K0
      LD      B13E3
      AND     M20019
      AND=    D30404 K0
      AND<>   D30403 K0
      ORB
      LD>     D30405 K405
      AND=    D30406 K0
      AND     B1022
      ORB
      LD      B1576
      AND=    D30405 K0
      AND<>   D30404 K0
      ORB
      ANB
      ORB
      OUT     M20063
1927  LDF     B13E3
      AND     M20019
      AND     B13FF
      AND<>   D30403 K0
      MOV     D30403 D30404
      MOV     K0 D30403
1938  LDF     B1576
      AND     M20063
      AND     B13FF
      AND<>   D30404 K0
      MOV     D30404 D30405
      MOV     K0 D30404
1949  LD      B13F7
      AND     B13FE
      OUT     M20163
1952  LD>=    D30405 K401
      AND<=   D30405 K409
      OR>=    D30405 K801
      OUT     B1022
1962  LD>=    D30405 K501
      AND<=   D30405 K511
      OUT     B1023
1969  LD      B13F8
      AND     B13FE
      LD      B13FF
      LD>     D30406 K406
      AND=    D30407 K0
      LD      B13E4
      AND     M20063
      AND=    D30406 K0
      AND<>   D30405 K0
      AND     B1022
      ORB
      ANB
      ORB
      OUT     M20020
1991  LDF     B13E4
      AND     M20063
      AND     B13FF
      AND<>   D30405 K0
      MOV     D30405 D30406
      MOV     K0 D30405
2002  LD      B13F9
      AND     B13FE
      OUT     M20120
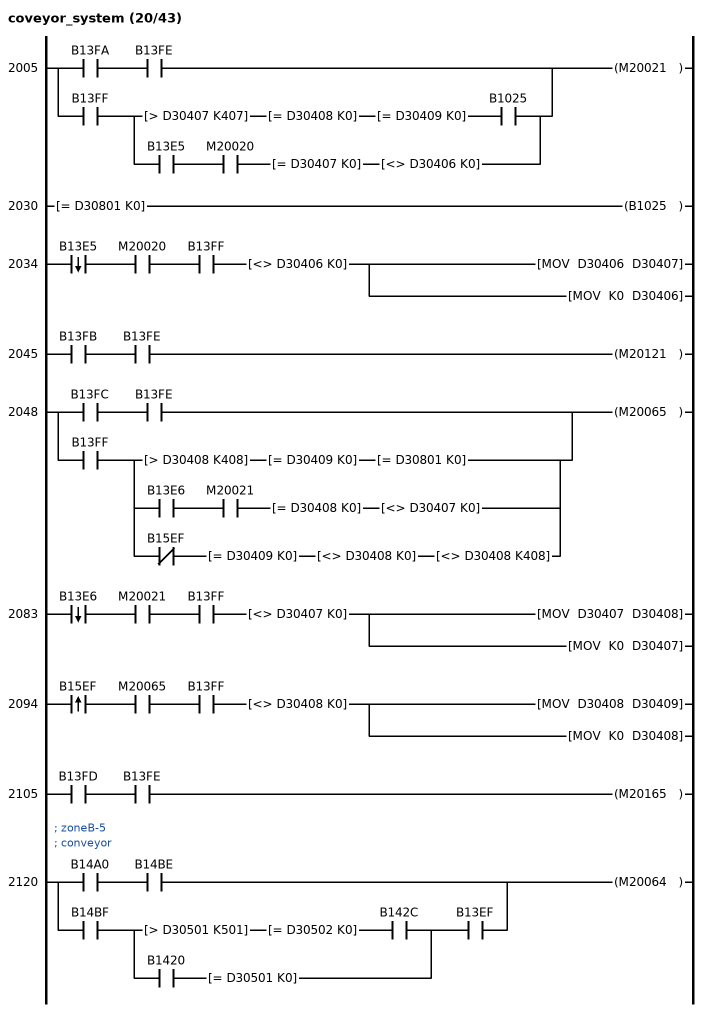
2005  LD      B13FA
      AND     B13FE
      LD      B13FF
      LD>     D30407 K407
      AND=    D30408 K0
      AND=    D30409 K0
      AND     B1025
      LD      B13E5
      AND     M20020
      AND=    D30407 K0
      AND<>   D30406 K0
      ORB
      ANB
      ORB
      OUT     M20021
2030  LD=     D30801 K0
      OUT     B1025
2034  LDF     B13E5
      AND     M20020
      AND     B13FF
      AND<>   D30406 K0
      MOV     D30406 D30407
      MOV     K0 D30406
2045  LD      B13FB
      AND     B13FE
      OUT     M20121
2048  LD      B13FC
      AND     B13FE
      LD      B13FF
      LD>     D30408 K408
      AND=    D30409 K0
      AND=    D30801 K0
      LD      B13E6
      AND     M20021
      AND=    D30408 K0
      AND<>   D30407 K0
      ORB
      LDI     B15EF
      AND=    D30409 K0
      AND<>   D30408 K0
      AND<>   D30408 K408
      ORB
      ANB
      ORB
      OUT     M20065
2083  LDF     B13E6
      AND     M20021
      AND     B13FF
      AND<>   D30407 K0
      MOV     D30407 D30408
      MOV     K0 D30407
2094  LDP     B15EF
      AND     M20065
      AND     B13FF
      AND<>   D30408 K0
      MOV     D30408 D30409
      MOV     K0 D30408
2105  LD      B13FD
      AND     B13FE
      OUT     M20165
; zoneB-5
; conveyor
2120  LD      B14A0
      AND     B14BE
      LD      B14BF
      LD>     D30501 K501
      AND=    D30502 K0
      AND     B142C
      LD      B1420
      AND=    D30501 K0
      ORB
      ANB
      AND     B13EF
      ORB
      OUT     M20064
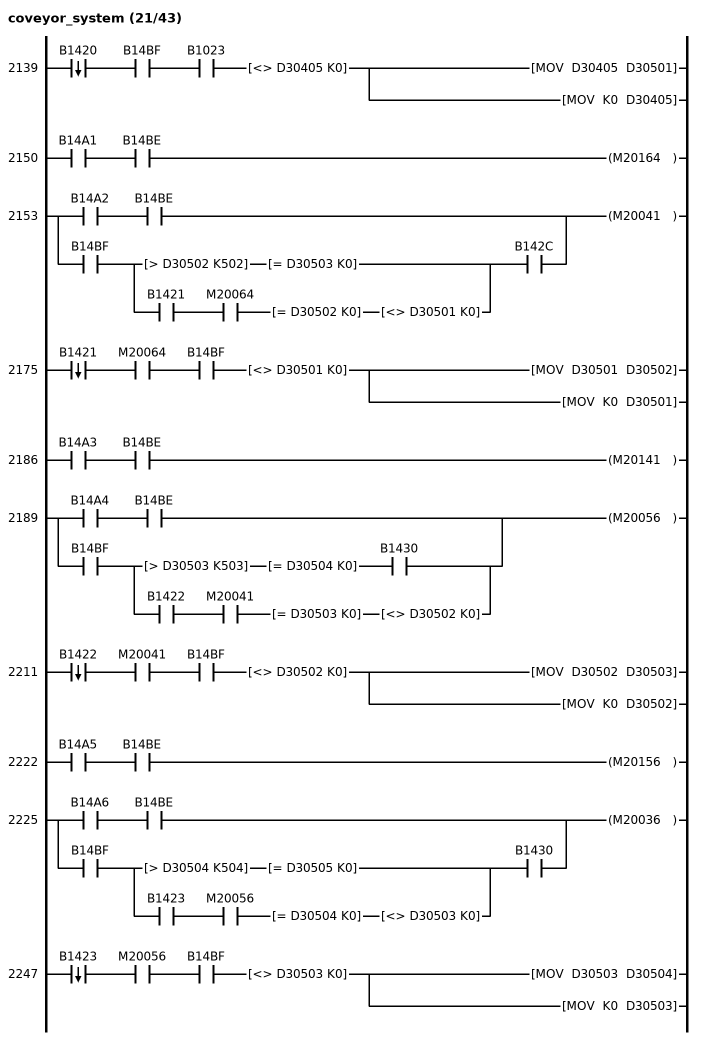
2139  LDF     B1420
      AND     B14BF
      AND     B1023
      AND<>   D30405 K0
      MOV     D30405 D30501
      MOV     K0 D30405
2150  LD      B14A1
      AND     B14BE
      OUT     M20164
2153  LD      B14A2
      AND     B14BE
      LD      B14BF
      LD>     D30502 K502
      AND=    D30503 K0
      LD      B1421
      AND     M20064
      AND=    D30502 K0
      AND<>   D30501 K0
      ORB
      ANB
      AND     B142C
      ORB
      OUT     M20041
2175  LDF     B1421
      AND     M20064
      AND     B14BF
      AND<>   D30501 K0
      MOV     D30501 D30502
      MOV     K0 D30501
2186  LD      B14A3
      AND     B14BE
      OUT     M20141
2189  LD      B14A4
      AND     B14BE
      LD      B14BF
      LD>     D30503 K503
      AND=    D30504 K0
      AND     B1430
      LD      B1422
      AND     M20041
      AND=    D30503 K0
      AND<>   D30502 K0
      ORB
      ANB
      ORB
      OUT     M20056
2211  LDF     B1422
      AND     M20041
      AND     B14BF
      AND<>   D30502 K0
      MOV     D30502 D30503
      MOV     K0 D30502
2222  LD      B14A5
      AND     B14BE
      OUT     M20156
2225  LD      B14A6
      AND     B14BE
      LD      B14BF
      LD>     D30504 K504
      AND=    D30505 K0
      LD      B1423
      AND     M20056
      AND=    D30504 K0
      AND<>   D30503 K0
      ORB
      ANB
      AND     B1430
      ORB
      OUT     M20036
2247  LDF     B1423
      AND     M20056
      AND     B14BF
      AND<>   D30503 K0
      MOV     D30503 D30504
      MOV     K0 D30503
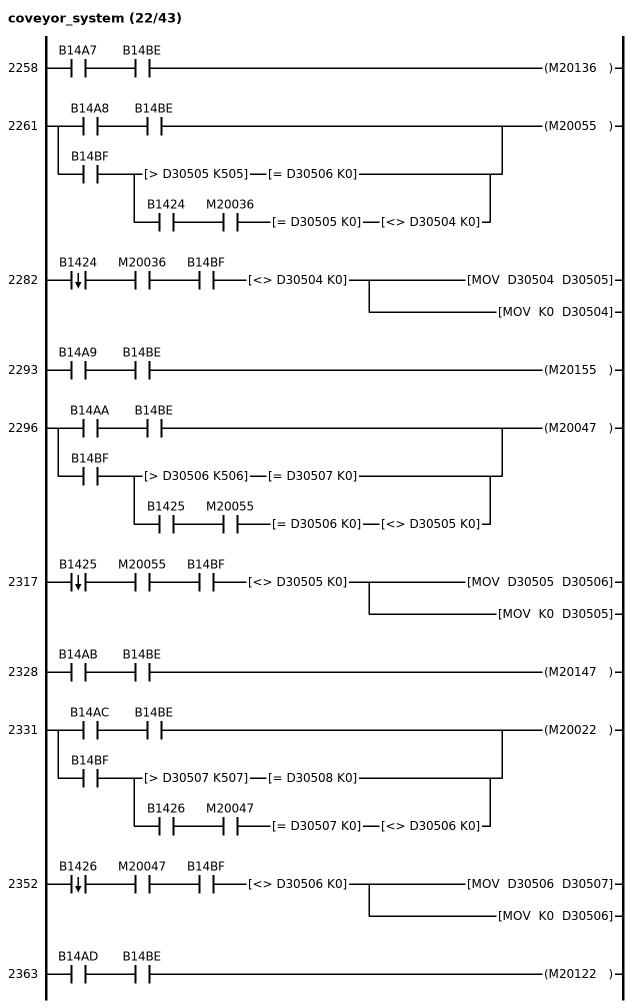
2258  LD      B14A7
      AND     B14BE
      OUT     M20136
2261  LD      B14A8
      AND     B14BE
      LD      B14BF
      LD>     D30505 K505
      AND=    D30506 K0
      LD      B1424
      AND     M20036
      AND=    D30505 K0
      AND<>   D30504 K0
      ORB
      ANB
      ORB
      OUT     M20055
2282  LDF     B1424
      AND     M20036
      AND     B14BF
      AND<>   D30504 K0
      MOV     D30504 D30505
      MOV     K0 D30504
2293  LD      B14A9
      AND     B14BE
      OUT     M20155
2296  LD      B14AA
      AND     B14BE
      LD      B14BF
      LD>     D30506 K506
      AND=    D30507 K0
      LD      B1425
      AND     M20055
      AND=    D30506 K0
      AND<>   D30505 K0
      ORB
      ANB
      ORB
      OUT     M20047
2317  LDF     B1425
      AND     M20055
      AND     B14BF
      AND<>   D30505 K0
      MOV     D30505 D30506
      MOV     K0 D30505
2328  LD      B14AB
      AND     B14BE
      OUT     M20147
2331  LD      B14AC
      AND     B14BE
      LD      B14BF
      LD>     D30507 K507
      AND=    D30508 K0
      LD      B1426
      AND     M20047
      AND=    D30507 K0
      AND<>   D30506 K0
      ORB
      ANB
      ORB
      OUT     M20022
2352  LDF     B1426
      AND     M20047
      AND     B14BF
      AND<>   D30506 K0
      MOV     D30506 D30507
      MOV     K0 D30506
2363  LD      B14AD
      AND     B14BE
      OUT     M20122
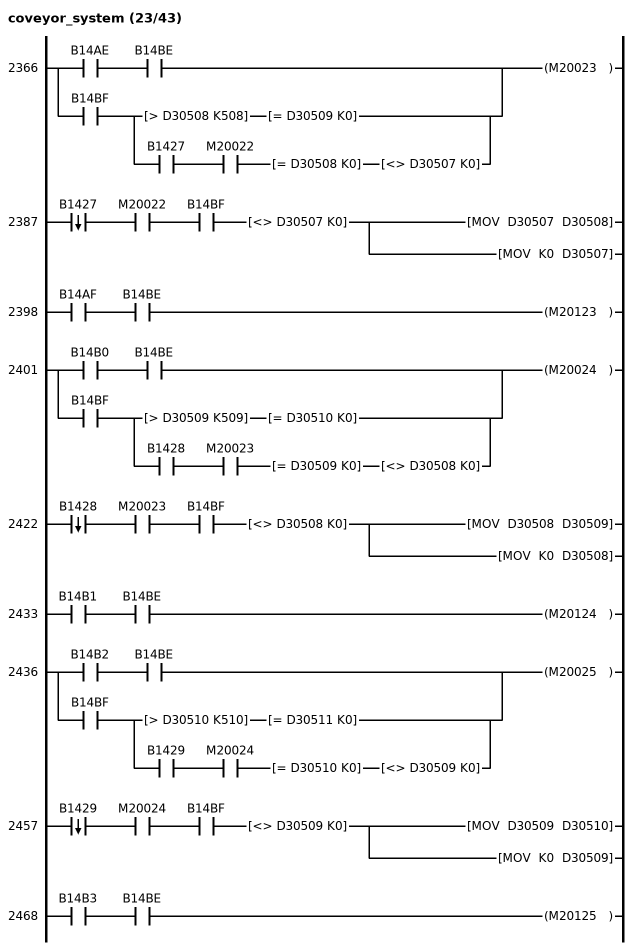
2366  LD      B14AE
      AND     B14BE
      LD      B14BF
      LD>     D30508 K508
      AND=    D30509 K0
      LD      B1427
      AND     M20022
      AND=    D30508 K0
      AND<>   D30507 K0
      ORB
      ANB
      ORB
      OUT     M20023
2387  LDF     B1427
      AND     M20022
      AND     B14BF
      AND<>   D30507 K0
      MOV     D30507 D30508
      MOV     K0 D30507
2398  LD      B14AF
      AND     B14BE
      OUT     M20123
2401  LD      B14B0
      AND     B14BE
      LD      B14BF
      LD>     D30509 K509
      AND=    D30510 K0
      LD      B1428
      AND     M20023
      AND=    D30509 K0
      AND<>   D30508 K0
      ORB
      ANB
      ORB
      OUT     M20024
2422  LDF     B1428
      AND     M20023
      AND     B14BF
      AND<>   D30508 K0
      MOV     D30508 D30509
      MOV     K0 D30508
2433  LD      B14B1
      AND     B14BE
      OUT     M20124
2436  LD      B14B2
      AND     B14BE
      LD      B14BF
      LD>     D30510 K510
      AND=    D30511 K0
      LD      B1429
      AND     M20024
      AND=    D30510 K0
      AND<>   D30509 K0
      ORB
      ANB
      ORB
      OUT     M20025
2457  LDF     B1429
      AND     M20024
      AND     B14BF
      AND<>   D30509 K0
      MOV     D30509 D30510
      MOV     K0 D30509
2468  LD      B14B3
      AND     B14BE
      OUT     M20125
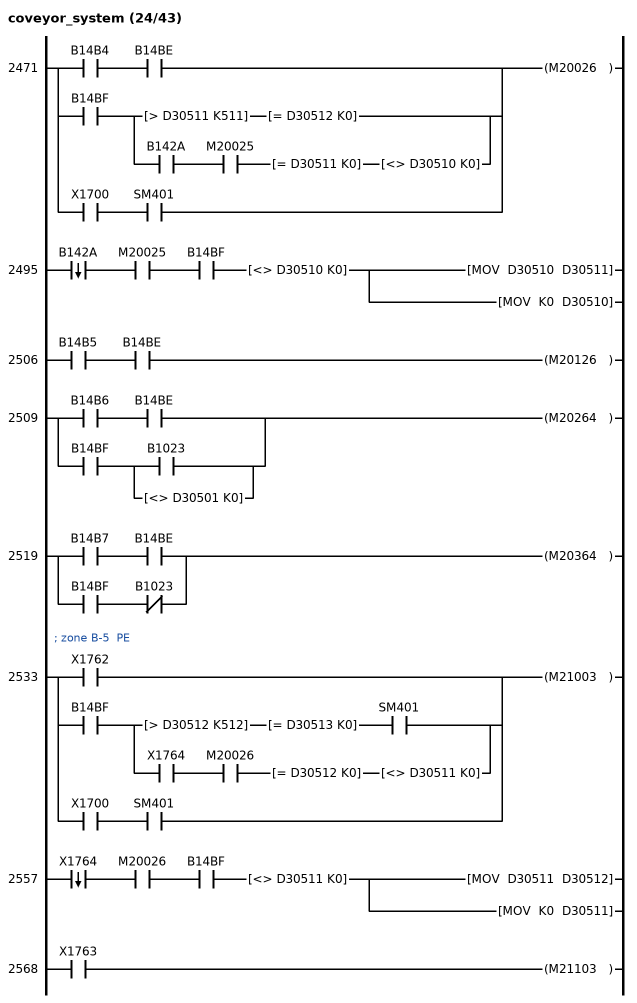
2471  LD      B14B4
      AND     B14BE
      LD      B14BF
      LD>     D30511 K511
      AND=    D30512 K0
      LD      B142A
      AND     M20025
      AND=    D30511 K0
      AND<>   D30510 K0
      ORB
      ANB
      ORB
      LD      X1700
      AND     SM401
      ORB
      OUT     M20026
2495  LDF     B142A
      AND     M20025
      AND     B14BF
      AND<>   D30510 K0
      MOV     D30510 D30511
      MOV     K0 D30510
2506  LD      B14B5
      AND     B14BE
      OUT     M20126
2509  LD      B14B6
      AND     B14BE
      LD      B14BF
      LD      B1023
      OR<>    D30501 K0
      ANB
      ORB
      OUT     M20264
2519  LD      B14B7
      AND     B14BE
      LD      B14BF
      ANI     B1023
      ORB
      OUT     M20364
; zone B-5  PE
2533  LD      X1762
      LD      B14BF
      LD>     D30512 K512
      AND=    D30513 K0
      AND     SM401
      LD      X1764
      AND     M20026
      AND=    D30512 K0
      AND<>   D30511 K0
      ORB
      ANB
      ORB
      LD      X1700
      AND     SM401
      ORB
      OUT     M21003
2557  LDF     X1764
      AND     M20026
      AND     B14BF
      AND<>   D30511 K0
      MOV     D30511 D30512
      MOV     K0 D30511
2568  LD      X1763
      OUT     M21103
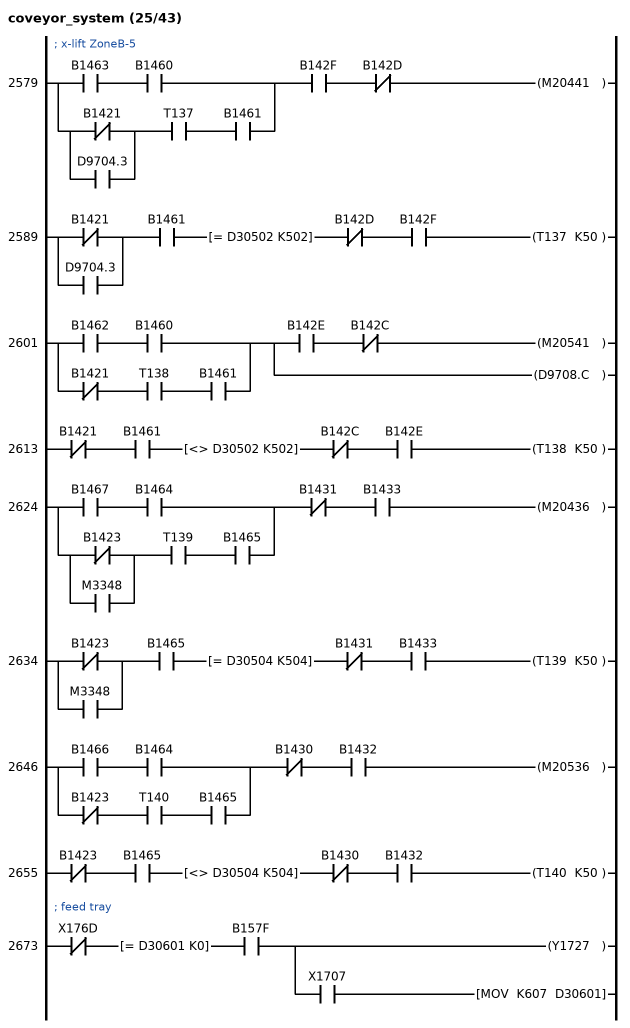
; x-lift ZoneB-5
2579  LD      B1463
      AND     B1460
      LDI     B1421
      OR      D9704.3
      AND     T137
      AND     B1461
      ORB
      AND     B142F
      ANI     B142D
      OUT     M20441
2589  LDI     B1421
      OR      D9704.3
      AND     B1461
      AND=    D30502 K502
      ANI     B142D
      AND     B142F
      OUT     T137 K50
2601  LD      B1462
      AND     B1460
      LDI     B1421
      AND     T138
      AND     B1461
      ORB
      MPS
      AND     B142E
      ANI     B142C
      OUT     M20541
      MPP
      OUT     D9708.C
2613  LDI     B1421
      AND     B1461
      AND<>   D30502 K502
      ANI     B142C
      AND     B142E
      OUT     T138 K50
2624  LD      B1467
      AND     B1464
      LDI     B1423
      OR      M3348
      AND     T139
      AND     B1465
      ORB
      ANI     B1431
      AND     B1433
      OUT     M20436
2634  LDI     B1423
      OR      M3348
      AND     B1465
      AND=    D30504 K504
      ANI     B1431
      AND     B1433
      OUT     T139 K50
2646  LD      B1466
      AND     B1464
      LDI     B1423
      AND     T140
      AND     B1465
      ORB
      ANI     B1430
      AND     B1432
      OUT     M20536
2655  LDI     B1423
      AND     B1465
      AND<>   D30504 K504
      ANI     B1430
      AND     B1432
      OUT     T140 K50
; feed tray
2673  LDI     X176D
      AND=    D30601 K0
      AND     B157F
      OUT     Y1727
      AND     X1707
      MOV     K607 D30601
